TYPE T_SnappyVerifyPort : UINT (25000..25999); END_TYPE

(* stored: Version 1.1.0.1, ProductVersion 3.1.4026.18
   DUT T_SnappyVerifyPort: Id {ad23866f-ec03-4546-9c4d-8b82ab63f61d} *)
